SYSTEM washer_detector
  (* Version 1.0, 2024-11-25, obotnar *)
  APPLICATION washer_detectorApp
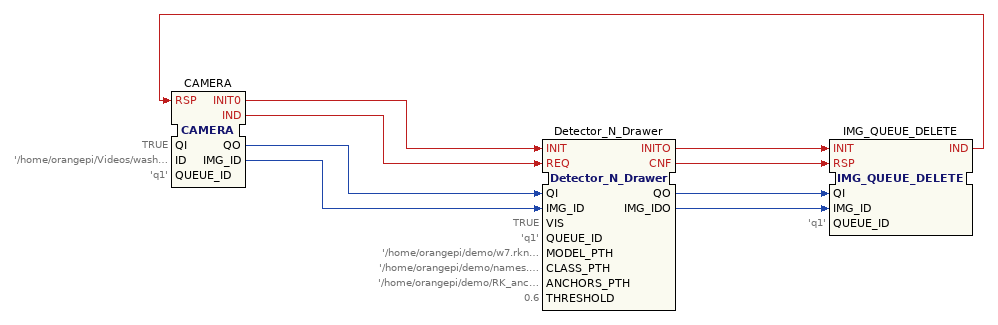
    FBS
      CAMERA : CAMERA(QI := TRUE, ID := '/home/orangepi/Videos/washer.webm', QUEUE_ID := 'q1');
      IMG_QUEUE_DELETE : IMG_QUEUE_DELETE(QUEUE_ID := 'q1');
      Detector_N_Drawer : Detector_N_Drawer(VIS := TRUE, QUEUE_ID := 'q1', MODEL_PTH := '/home/orangepi/demo/w7.rknn', CLASS_PTH := '/home/orangepi/demo/names.txt', ANCHORS_PTH := '/home/orangepi/demo/RK_anchors.txt', THRESHOLD := 0.6);
    END_FBS
    EVENT_CONNECTIONS
      CAMERA.INIT0 TO Detector_N_Drawer.INIT;
      CAMERA.IND TO Detector_N_Drawer.REQ;
      Detector_N_Drawer.INITO TO IMG_QUEUE_DELETE.INIT;
      Detector_N_Drawer.CNF TO IMG_QUEUE_DELETE.RSP;
      IMG_QUEUE_DELETE.IND TO CAMERA.RSP;
    END_CONNECTIONS
    DATA_CONNECTIONS
      Detector_N_Drawer.QO TO IMG_QUEUE_DELETE.QI;
      Detector_N_Drawer.IMG_IDO TO IMG_QUEUE_DELETE.IMG_ID;
      CAMERA.QO TO Detector_N_Drawer.QI;
      CAMERA.IMG_ID TO Detector_N_Drawer.IMG_ID;
    END_CONNECTIONS
  END_APPLICATION
  DEVICE FORTE_PC : FORTE_PC(MGR_ID := "10.5.20.198:61499" (* Device manager socket ID *))
    {SET_ATTRIBUTE(Profile, HOLOBLOC)}
    RESOURCE EMB_RES : EMB_RES
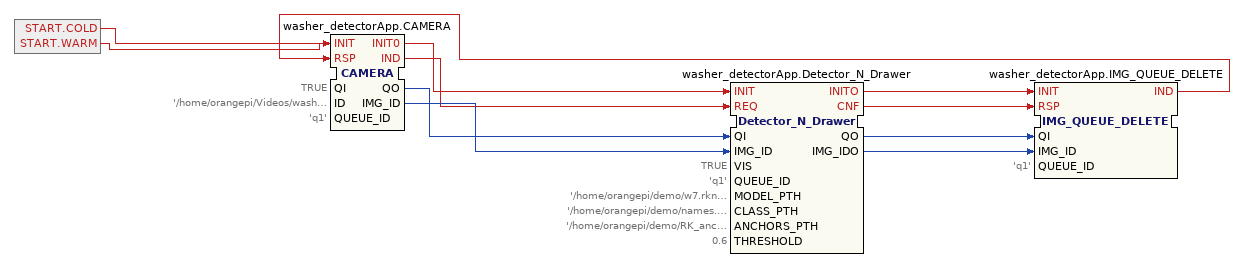
      FBS
        washer_detectorApp.CAMERA : CAMERA(QI := TRUE, ID := '/home/orangepi/Videos/washer.webm', QUEUE_ID := 'q1');
        washer_detectorApp.IMG_QUEUE_DELETE : IMG_QUEUE_DELETE(QUEUE_ID := 'q1');
        washer_detectorApp.Detector_N_Drawer : Detector_N_Drawer(VIS := TRUE, QUEUE_ID := 'q1', MODEL_PTH := '/home/orangepi/demo/w7.rknn', CLASS_PTH := '/home/orangepi/demo/names.txt', ANCHORS_PTH := '/home/orangepi/demo/RK_anchors.txt', THRESHOLD := 0.6);
      END_FBS
      EVENT_CONNECTIONS
        START.COLD TO washer_detectorApp.CAMERA.INIT;
        START.WARM TO washer_detectorApp.CAMERA.INIT;
        washer_detectorApp.CAMERA.INIT0 TO washer_detectorApp.Detector_N_Drawer.INIT;
        washer_detectorApp.CAMERA.IND TO washer_detectorApp.Detector_N_Drawer.REQ;
        washer_detectorApp.Detector_N_Drawer.INITO TO washer_detectorApp.IMG_QUEUE_DELETE.INIT;
        washer_detectorApp.Detector_N_Drawer.CNF TO washer_detectorApp.IMG_QUEUE_DELETE.RSP;
        washer_detectorApp.IMG_QUEUE_DELETE.IND TO washer_detectorApp.CAMERA.RSP;
      END_CONNECTIONS
      DATA_CONNECTIONS
        washer_detectorApp.CAMERA.QO TO washer_detectorApp.Detector_N_Drawer.QI;
        washer_detectorApp.CAMERA.IMG_ID TO washer_detectorApp.Detector_N_Drawer.IMG_ID;
        washer_detectorApp.Detector_N_Drawer.QO TO washer_detectorApp.IMG_QUEUE_DELETE.QI;
        washer_detectorApp.Detector_N_Drawer.IMG_IDO TO washer_detectorApp.IMG_QUEUE_DELETE.IMG_ID;
      END_CONNECTIONS
    END_RESOURCE
  END_DEVICE
  MAPPINGS
    washer_detectorApp.CAMERA ON FORTE_PC.EMB_RES;
    washer_detectorApp.IMG_QUEUE_DELETE ON FORTE_PC.EMB_RES;
    washer_detectorApp.Detector_N_Drawer ON FORTE_PC.EMB_RES;
  END_MAPPINGS
  SEGMENTS
    Ethernet : Ethernet;
  END_SEGMENTS
  LINKS
    FORTE_PC => Ethernet;
  END_LINKS
END_SYSTEM
